# EPICS autosave request: autosave/galil_reverse_transforms.req
$(P)$(M)_RTRANSFORMA_SP
$(P)$(M)_RTRANSFORMB_SP
$(P)$(M)_RTRANSFORMC_SP
$(P)$(M)_RTRANSFORMD_SP
$(P)$(M)_RTRANSFORME_SP
$(P)$(M)_RTRANSFORMF_SP
$(P)$(M)_RTRANSFORMG_SP
$(P)$(M)_RTRANSFORMH_SP
